# EPICS substitutions: evrSupport/Db/ioc/bsaXL03.substitutions
#####################
# BSA functionality for devices
# load these for sim or real data
####################
# BSA records
# One per device:
#
file bsaBPMSEdef.db {
  pattern {DEVICE      , LOC  , UN, SYS, SLCLNK }
	  { BPMS:XX03:1, IN20,EV02, SYS0, "BPMS:XX03:1:FANOUTSLC PP"}
	  { BPMS:XX03:2, IN20,EV02, SYS0, "BPMS:XX03:2:FANOUTSLC PP"}
	  { BPMS:XX03:3, IN20,EV02, SYS0, "BPMS:XX03:3:FANOUTSLC PP"}
	  { BPMS:XX03:4, IN20,EV02, SYS0, "BPMS:XX03:4:FANOUTSLC PP"}
	  { BPMS:XX03:5, IN20,EV02, SYS0, "BPMS:XX03:5:FANOUTSLC PP"}
	  { BPMS:XX03:6, IN20,EV02, SYS0, "BPMS:XX03:6:FANOUTSLC PP"}
}

file bsaTOROEdef.db {
  pattern {DEVICE       , LOC , UN , SYS, SLCLNK }
	  { TORO:XX03:1 ,IN20 ,EV02, SYS0, "TORO:XX03:1:FANOUTSLC PP"}
	  { TORO:XX03:2 ,IN20 ,EV02, SYS0, "TORO:XX03:2:FANOUTSLC PP"}
}
file bsaPMTEdef.db {
  pattern {DEVICE      , LOC , UN , SYS, SLCLNK  }
	  { PMT:XX03:1 , IN20,EV02, SYS0, "PMT:XX03:1:FANOUTSLC PP"}
	  { PMT:XX03:2 , IN20,EV02, SYS0, "PMT:XX03:2:FANOUTSLC PP"}
	  { PMT:XX03:3 , IN20,EV02, SYS0, "PMT:XX03:3:FANOUTSLC PP"}
	  { PMT:XX03:4 , IN20,EV02, SYS0, "PMT:XX03:4:FANOUTSLC PP"}
	  { PMT:XX03:5 , IN20,EV02, SYS0, "PMT:XX03:5:FANOUTSLC PP"}
	  { PMT:XX03:6 , IN20,EV02, SYS0, "PMT:XX03:6:FANOUTSLC PP"}
}
file bsaBLENEdef.db {
  pattern {DEVICE       , LOC , UN , SYS, SLCLNK  }
	  { BLEN:XX03:1 , IN20,EV02, SYS0, "BLEN:XX03:1:FANOUTSLC PP"}
	  { BLEN:XX03:2 , IN20,EV02, SYS0, "BLEN:XX03:2:FANOUTSLC PP"}
	  { BLEN:XX03:3 , IN20,EV02, SYS0, "BLEN:XX03:3:FANOUTSLC PP"}
}
file bsaWIREEdef.db {
  pattern {DEVICE       , LOC , UN , SYS, SLCLNK  }
	  { WIRE:XX03:1 , IN20,EV02, SYS0, "WIRE:XX03:1:FANOUTSLC PP"}
	  { WIRE:XX03:2 , IN20,EV02, SYS0, "WIRE:XX03:2:FANOUTSLC PP"}
	  { WIRE:XX03:3 , IN20,EV02, SYS0, "WIRE:XX03:3:FANOUTSLC PP"}
	  { WIRE:XX03:4 , IN20,EV02, SYS0, "WIRE:XX03:4:FANOUTSLC PP"}
}
